FUNCTION_BLOCK Mux
  (* Version 1.0, 2007-08-28, Goran Cengic, Chalmers *)
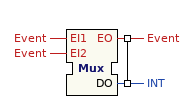
  EVENT_INPUT
    EI1;
    EI2;
  END_EVENT
  EVENT_OUTPUT
    EO WITH DO;
  END_EVENT
  VAR_OUTPUT
    DO : INT;
  END_VAR
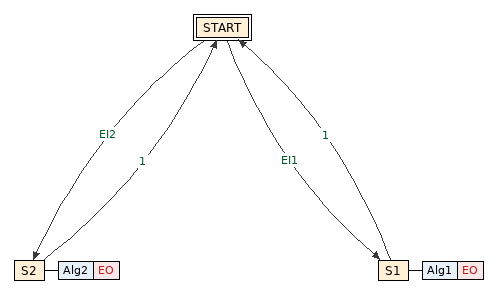
  EC_STATES
    START;
    S1 : Alg1 -> EO;
    S2 : Alg2 -> EO;
  END_STATES
  EC_TRANSITIONS
    START TO S1 := EI1;
    S1 TO START := 1;
    START TO S2 := EI2;
    S2 TO START := 1;
  END_TRANSITIONS
  ALGORITHM Alg1 IN Java:
DO = 1;
  END_ALGORITHM
  ALGORITHM Alg2 IN Java:
DO = 2;
  END_ALGORITHM
END_FUNCTION_BLOCK
